Staubli VAL3: clkValve16.pgx

program clkValve16()
begin
  call toggleValve(16)
end
